FUNCTION_BLOCK CmdVent (* CAT Function Block Type *)
  (* Standard: 61499-2 *)
  (* Version 0.0, 6/7/2026, Schneider Electric, template *)
  PACKAGE SE.Nereda;
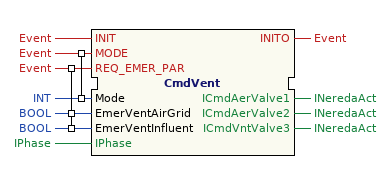
  EVENT_INPUT
    INIT;
    MODE WITH Mode;
    REQ_EMER_PAR WITH EmerVentAirGrid, EmerVentInfluent;
  END_EVENT
  EVENT_OUTPUT
    INITO;
  END_EVENT
  VAR_INPUT
    Mode : INT;
    EmerVentAirGrid : BOOL;
    EmerVentInfluent : BOOL;
  END_VAR
  SOCKETS
    IPhase : IPhase;
  END_SOCKETS
  PLUGS
    ICmdAerValve1 : INeredaAct;
    ICmdAerValve2 : INeredaAct;
    ICmdVntValve3 : INeredaAct;
  END_PLUGS
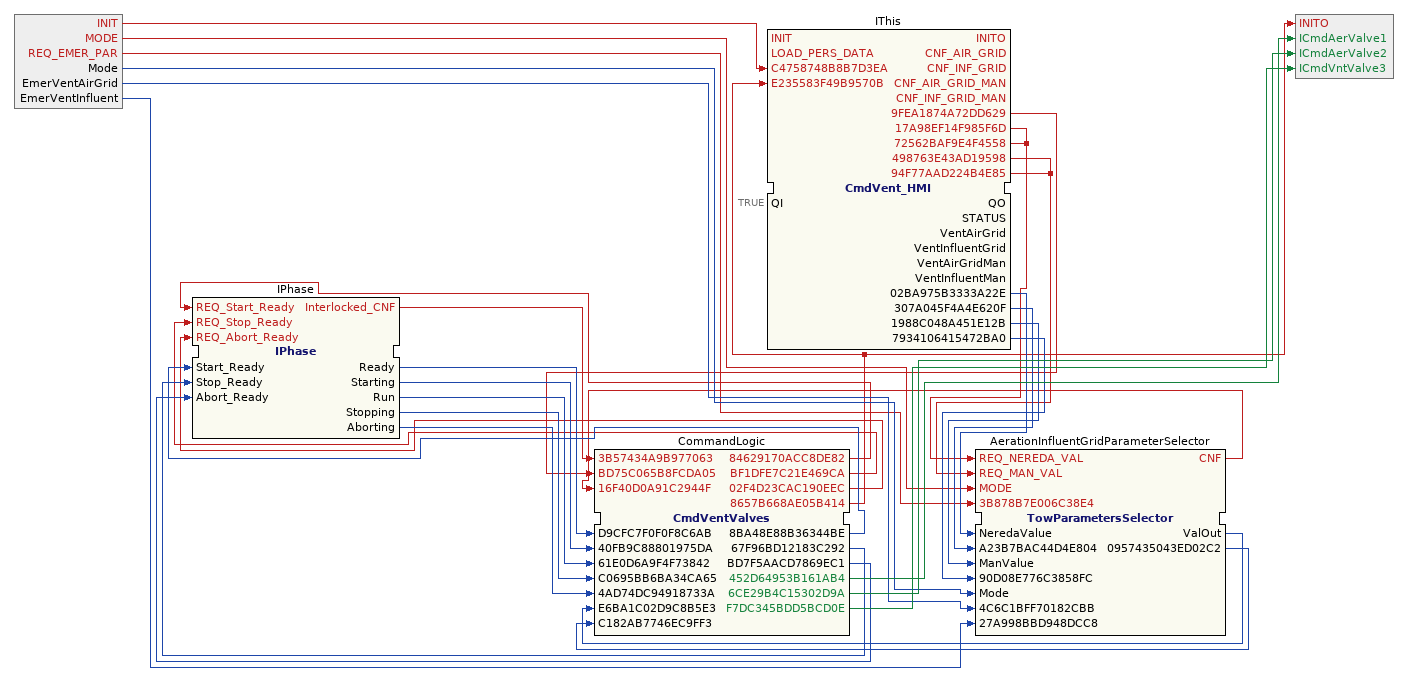
  (* 01 - FUNCTIONNAL INPUT INTERFACE *)
  (* 00 - INITIALIZATION *)
  (* 05 - LOGIC *)
  (* 06 - HMI INTERFACE *)
  (* 03 - FIELD INTERFACE *)
  (* 02 - FUNCTIONNAL OUTPUT INTERFACE *)
  (* Command Logic *)
  (* Parameters Setpoint *)
  FBS
    IThis : CmdVent_HMI(QI := TRUE);
    CommandLogic : CmdVentValves; {SET_ATTRIBUTE(Configuration.Component.HideUnusedPorts, )}
    AerationInfluentGridParameterSelector : TowParametersSelector;
  END_FBS
  EVENT_CONNECTIONS
    INIT TO IThis.C4758748B8B7D3EA;
    IPhase.Interlocked_CNF TO CommandLogic.3B57434A9B977063;
    CommandLogic.84629170ACC8DE82 TO IPhase.REQ_Start_Ready;
    CommandLogic.BF1DFE7C21E469CA TO IPhase.REQ_Stop_Ready;
    CommandLogic.02F4D23CAC190EEC TO IPhase.REQ_Abort_Ready;
    IThis.9FEA1874A72DD629 TO CommandLogic.BD75C065B8FCDA05;
    CommandLogic.8657B668AE05B414 TO INITO;
    CommandLogic.8657B668AE05B414 TO IThis.E235583F49B9570B;
    AerationInfluentGridParameterSelector.CNF TO CommandLogic.16F40D0A91C2944F;
    IThis.17A98EF14F985F6D TO AerationInfluentGridParameterSelector.REQ_NEREDA_VAL;
    IThis.72562BAF9E4F4558 TO AerationInfluentGridParameterSelector.REQ_NEREDA_VAL;
    IThis.498763E43AD19598 TO AerationInfluentGridParameterSelector.REQ_MAN_VAL;
    IThis.94F77AAD224B4E85 TO AerationInfluentGridParameterSelector.REQ_MAN_VAL;
    MODE TO AerationInfluentGridParameterSelector.MODE;
    REQ_EMER_PAR TO AerationInfluentGridParameterSelector.3B878B7E006C38E4;
  END_CONNECTIONS
  DATA_CONNECTIONS
    IPhase.Ready TO CommandLogic.D9CFC7F0F0F8C6AB;
    IPhase.Starting TO CommandLogic.40FB9C88801975DA;
    IPhase.Run TO CommandLogic.61E0D6A9F4F73842;
    IPhase.Stopping TO CommandLogic.C0695BB6BA34CA65;
    IPhase.Aborting TO CommandLogic.4AD74DC94918733A;
    CommandLogic.8BA48E88B36344BE TO IPhase.Start_Ready;
    CommandLogic.67F96BD12183C292 TO IPhase.Stop_Ready;
    CommandLogic.BD7F5AACD7869EC1 TO IPhase.Abort_Ready;
    AerationInfluentGridParameterSelector.ValOut TO CommandLogic.E6BA1C02D9C8B5E3;
    AerationInfluentGridParameterSelector.0957435043ED02C2 TO CommandLogic.C182AB7746EC9FF3;
    IThis.02BA975B3333A22E TO AerationInfluentGridParameterSelector.NeredaValue;
    IThis.307A045F4A4E620F TO AerationInfluentGridParameterSelector.A23B7BAC44D4E804;
    IThis.1988C048A451E12B TO AerationInfluentGridParameterSelector.ManValue;
    IThis.7934106415472BA0 TO AerationInfluentGridParameterSelector.90D08E776C3858FC;
    Mode TO AerationInfluentGridParameterSelector.Mode;
    EmerVentAirGrid TO AerationInfluentGridParameterSelector.4C6C1BFF70182CBB;
    EmerVentInfluent TO AerationInfluentGridParameterSelector.27A998BBD948DCC8;
  END_CONNECTIONS
  ADAPTER_CONNECTIONS
    CommandLogic.452D64953B161AB4 TO ICmdAerValve1;
    CommandLogic.6CE29B4C15302D9A TO ICmdAerValve2;
    CommandLogic.F7DC345BDD5BCD0E TO ICmdVntValve3;
  END_CONNECTIONS
END_FUNCTION_BLOCK
